// TIA Portal V18 export
TYPE "User_data_type_1"
   STRUCT
      MoteurType { ExternalAccessible := 'False'; ExternalVisible := 'False'; ExternalWritable := 'False'} : Struct
         Enable : Bool;
         StartMode : DInt;
         StopMode : Int;
         Status : Bool;
         Busy : Bool;
         Error : Bool;
         ErrorId : Word;
      END_STRUCT;
   END_STRUCT;
END_TYPE
